PROGRAM EM03_Placing2
VAR
	
	//Backbone
	FB_StateMachine_Placing2		: FB_StateManager;
	bFl_RunningMachinePlacing2		: BOOL;
	bFl_SeqReset					: BOOL;
	bFl_Manual						: BOOL;
	CheckStatusPlacing2				: checkstatus;
	AlarmEventHistory				: ARRAY[1..20] OF Alarm_Event_History;
	Placing2_Management				: FB_Placing;
	bFl_Flushing					: BOOL;
	PalletID_Placing2				: PalletID_Name;
	Placing2_ID						: STRING;
	bFl_PalletJammed				: BOOL;
	
	//Motor
	Motor_PalletPlacing2			: MotorManagement;
	bFl_MotorPlacing2				: BOOL;
	Motor_Placing2_Error			: BOOL;
	Motor_Placing2_ErrorID			: UINT;
	bFl_MotorPlacing2_Fwd			: BOOL;
	bFl_MotorPlacing2_Rev			: BOOL;
	bFL_Safety						: BOOL;
	AlarmEventActive				: ARRAY[1..20] OF Alarm_Event_Active;
	CheckAcc						: TON;
END_VAR
VAR // added by the converter: edge detectors and wires of the graphical bodies
    _w1 : BOOL;
END_VAR

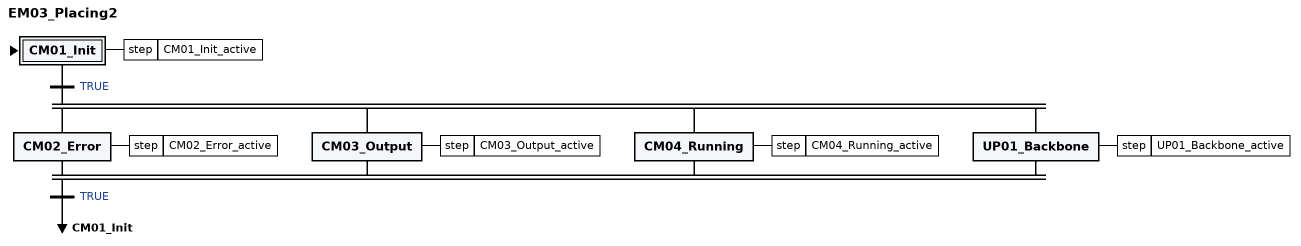
INITIAL_STEP CM01_Init:
    CM01_Init_active(N);  // step action
END_STEP
TRANSITION FROM CM01_Init TO (CM02_Error, CM03_Output, CM04_Running, UP01_Backbone)
    := TRUE;
END_TRANSITION
STEP CM02_Error:
    CM02_Error_active(N);  // step action
END_STEP
STEP CM03_Output:
    CM03_Output_active(N);  // step action
END_STEP
STEP CM04_Running:
    CM04_Running_active(N);  // step action
END_STEP
STEP UP01_Backbone:
    UP01_Backbone_active(N);  // step action
END_STEP
TRANSITION FROM (CM02_Error, CM03_Output, CM04_Running, UP01_Backbone) TO CM01_Init
    := TRUE;
END_TRANSITION

ACTION CM01_Init_active:
Data_GVL.bFL_StartPlacing2			:= Status_GVL.bFl_RunButton_Robotic OR HMI_GVL.bStartButtonPlacing2;
Data_GVL.bFL_StopPlacing2			:= NOT Status_GVL.bFl_StopButton_Robotic OR HMI_GVL.bStopButtonPlacing2;
Data_GVL.bFL_ResetPlacing2			:= Status_GVL.bFl_ResetButton_Robotic OR HMI_GVL.bResetButtonPlacing2;
Data_GVL.bFL_AckPlacing2			:= Status_GVL.bFl_Acknowledge_Robotic OR HMI_GVL.bAcknowledgeButtonPlacing2;
Data_GVL.bFL_AutoManuaModePlacing2 	:= Status_GVL.bFl_Manual_Robotic OR HMI_GVL.bTestModeEnablePlacing2;
bFl_RunningMachinePlacing2			:= Data_GVL.stStateMachinePlacing2.Running;
bFl_Manual							:= Data_GVL.stStateMachinePlacing2.ManualMode;
bFl_SeqReset						:= NOT Status_GVL.bFl_EStop_Robotic;
bFL_Safety							:= Status_GVL.bFl_EStop_Robotic AND Status_GVL.bSafety_DoorRobotic;


(*=================Convert Timer============================*)
Data_GVL.Tmr_Placing2	:= ConvertMilliSecTimeData(HMI_GVL.Tmr_Placing2);

(*=================Data OEE============================*)
Data_GVL.dt_Production[2].Data1			:= HMI_GVL.arCountTotal[2];
Data_GVL.dt_Production[2].Data2			:= HMI_GVL.arPalletTotal[2];
Data_GVL.dt_Production[2].Data3			:= HMI_GVL.arPalletIncomplete[2];
Data_GVL.dt_Production[2].ProductCode	:= Status_GVL.RecipeLine[2].ProductName;
END_ACTION

ACTION CM02_Error_active:
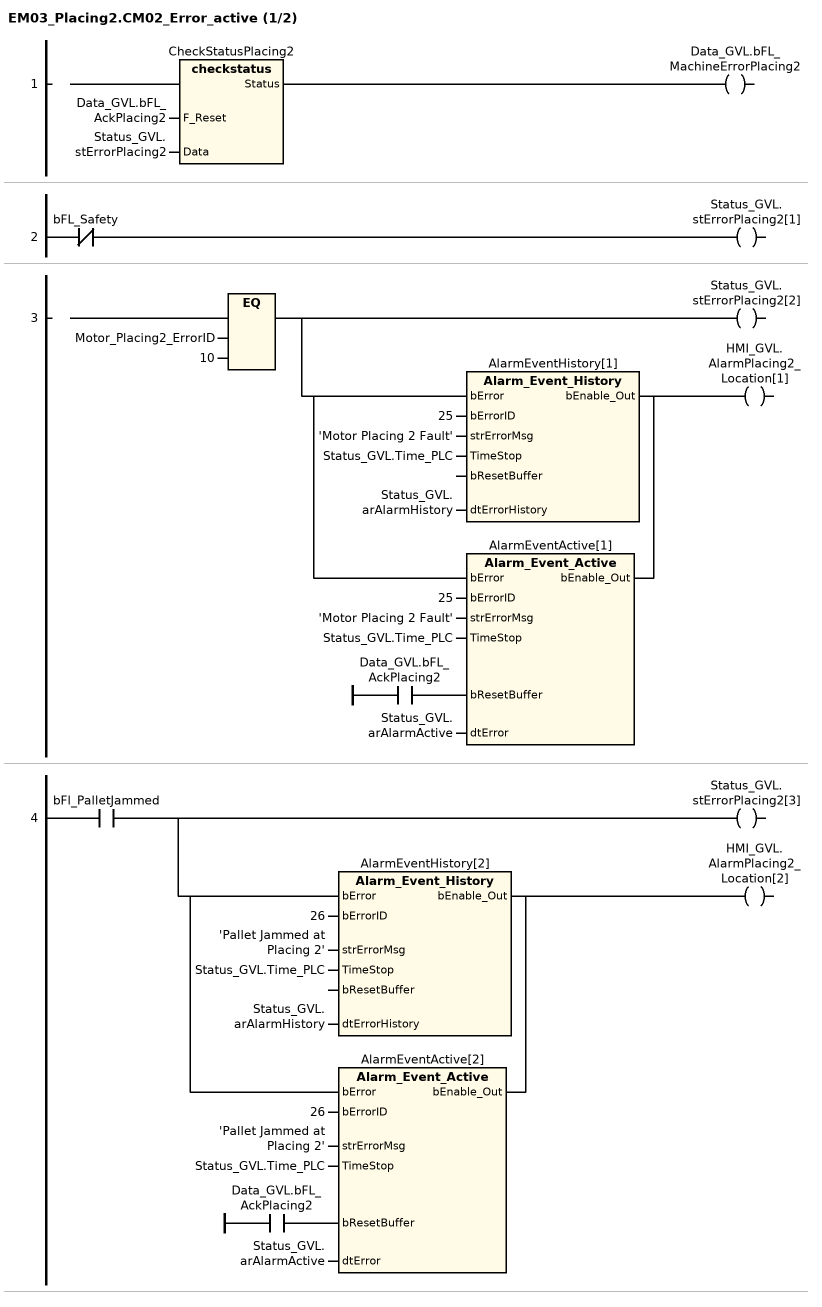
// NETWORK 1
CheckStatusPlacing2(F_Reset := Data_GVL.bFL_AckPlacing2, Data := Status_GVL.stErrorPlacing2); // checkstatus
Data_GVL.bFL_MachineErrorPlacing2 := CheckStatusPlacing2.Status;

// NETWORK 2
Status_GVL.stErrorPlacing2[1] := NOT bFL_Safety;

// NETWORK 3
_w1 := Motor_Placing2_ErrorID = 10;
Status_GVL.stErrorPlacing2[2] := _w1;
AlarmEventHistory[1](
    bError := _w1,
    bErrorID := 25,
    strErrorMsg := 'Motor Placing 2 Fault',
    TimeStop := Status_GVL.Time_PLC,
    dtErrorHistory := Status_GVL.arAlarmHistory); // Alarm_Event_History
AlarmEventActive[1](
    bError := _w1,
    bErrorID := 25,
    strErrorMsg := 'Motor Placing 2 Fault',
    TimeStop := Status_GVL.Time_PLC,
    bResetBuffer := Data_GVL.bFL_AckPlacing2,
    dtError := Status_GVL.arAlarmActive); // Alarm_Event_Active
HMI_GVL.AlarmPlacing2_Location[1] := AlarmEventHistory[1].bEnable_Out OR AlarmEventActive[1].bEnable_Out;

// NETWORK 4
Status_GVL.stErrorPlacing2[3] := bFl_PalletJammed;
AlarmEventHistory[2](
    bError := bFl_PalletJammed,
    bErrorID := 26,
    strErrorMsg := 'Pallet Jammed at Placing 2',
    TimeStop := Status_GVL.Time_PLC,
    dtErrorHistory := Status_GVL.arAlarmHistory); // Alarm_Event_History
AlarmEventActive[2](
    bError := bFl_PalletJammed,
    bErrorID := 26,
    strErrorMsg := 'Pallet Jammed at Placing 2',
    TimeStop := Status_GVL.Time_PLC,
    bResetBuffer := Data_GVL.bFL_AckPlacing2,
    dtError := Status_GVL.arAlarmActive); // Alarm_Event_Active
HMI_GVL.AlarmPlacing2_Location[2] := AlarmEventHistory[2].bEnable_Out OR AlarmEventActive[2].bEnable_Out;

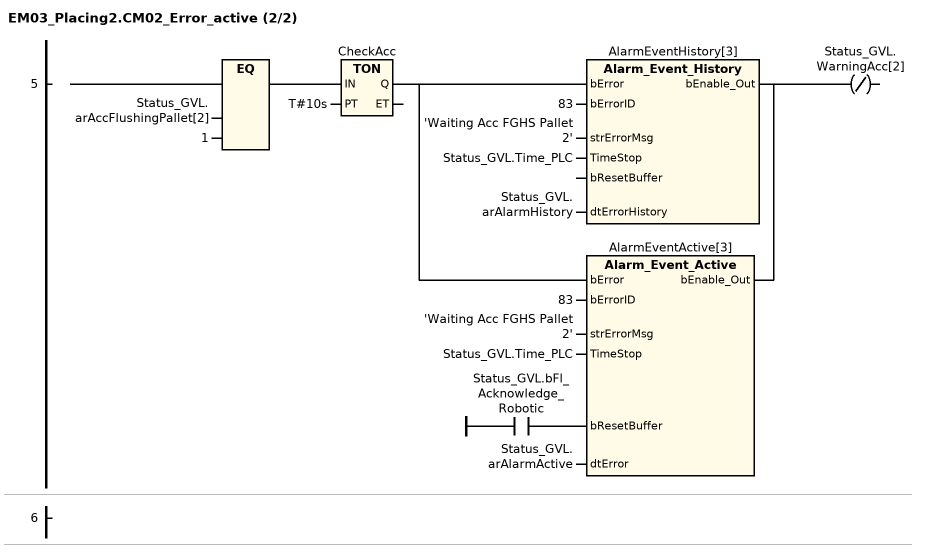
// NETWORK 5
CheckAcc(IN := Status_GVL.arAccFlushingPallet[2] = 1, PT := T#10s); // TON
AlarmEventHistory[3](
    bError := CheckAcc.Q,
    bErrorID := 83,
    strErrorMsg := 'Waiting Acc FGHS Pallet 2',
    TimeStop := Status_GVL.Time_PLC,
    dtErrorHistory := Status_GVL.arAlarmHistory); // Alarm_Event_History
AlarmEventActive[3](
    bError := CheckAcc.Q,
    bErrorID := 83,
    strErrorMsg := 'Waiting Acc FGHS Pallet 2',
    TimeStop := Status_GVL.Time_PLC,
    bResetBuffer := Status_GVL.bFl_Acknowledge_Robotic,
    dtError := Status_GVL.arAlarmActive); // Alarm_Event_Active
Status_GVL.WarningAcc[2] := NOT (AlarmEventHistory[3].bEnable_Out OR AlarmEventActive[3].bEnable_Out);

// NETWORK 6
END_ACTION

ACTION CM03_Output_active:
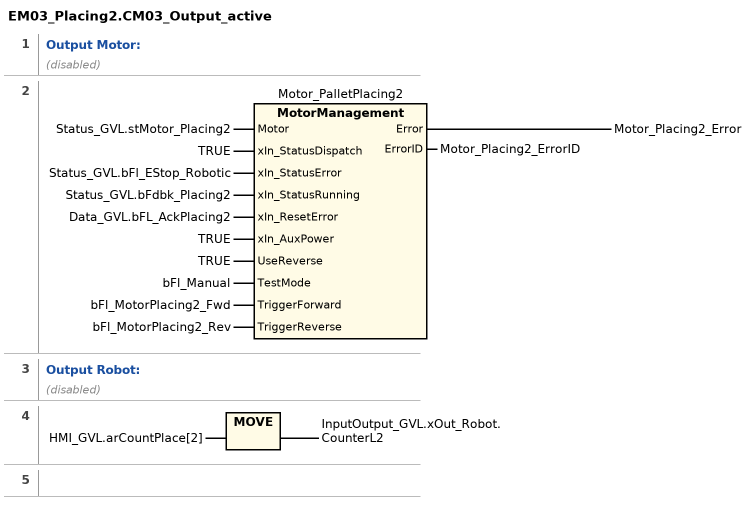
// NETWORK 1 (disabled)
// label: Output Motor

// NETWORK 2
Motor_PalletPlacing2(
    Motor := Status_GVL.stMotor_Placing2,
    xIn_StatusDispatch := TRUE,
    xIn_StatusError := Status_GVL.bFl_EStop_Robotic,
    xIn_StatusRunning := Status_GVL.bFdbk_Placing2,
    xIn_ResetError := Data_GVL.bFL_AckPlacing2,
    xIn_AuxPower := TRUE,
    UseReverse := TRUE,
    TestMode := bFl_Manual,
    TriggerForward := bFl_MotorPlacing2_Fwd,
    TriggerReverse := bFl_MotorPlacing2_Rev,
    ErrorID => Motor_Placing2_ErrorID); // MotorManagement
Motor_Placing2_Error := Motor_PalletPlacing2.Error;

// NETWORK 3 (disabled)
// label: Output Robot

// NETWORK 4
InputOutput_GVL.xOut_Robot.CounterL2 := HMI_GVL.arCountPlace[2];

// NETWORK 5
END_ACTION

ACTION CM04_Running_active:
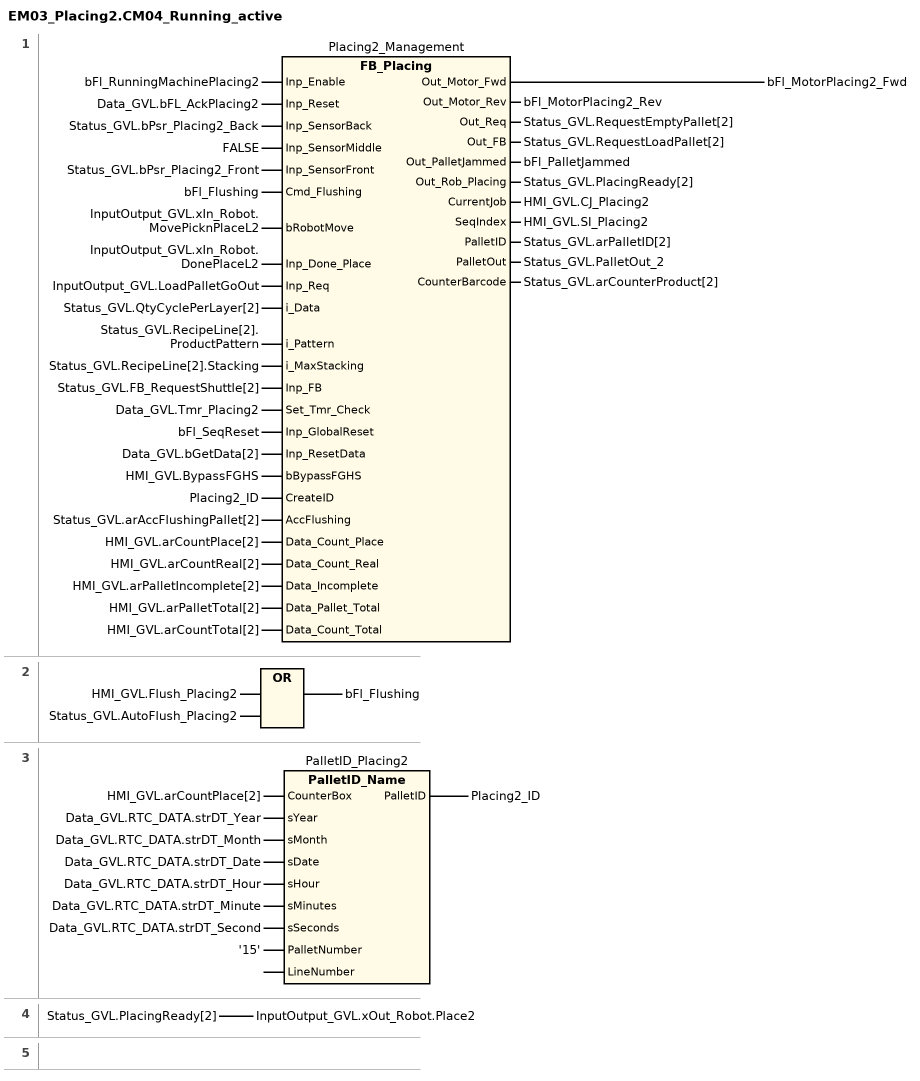
// NETWORK 1
Placing2_Management(
    Inp_Enable := bFl_RunningMachinePlacing2,
    Inp_Reset := Data_GVL.bFL_AckPlacing2,
    Inp_SensorBack := Status_GVL.bPsr_Placing2_Back,
    Inp_SensorMiddle := FALSE,
    Inp_SensorFront := Status_GVL.bPsr_Placing2_Front,
    Cmd_Flushing := bFl_Flushing,
    bRobotMove := InputOutput_GVL.xIn_Robot.MovePicknPlaceL2,
    Inp_Done_Place := InputOutput_GVL.xIn_Robot.DonePlaceL2,
    Inp_Req := InputOutput_GVL.LoadPalletGoOut,
    i_Data := Status_GVL.QtyCyclePerLayer[2],
    i_Pattern := Status_GVL.RecipeLine[2].ProductPattern,
    i_MaxStacking := Status_GVL.RecipeLine[2].Stacking,
    Inp_FB := Status_GVL.FB_RequestShuttle[2],
    Set_Tmr_Check := Data_GVL.Tmr_Placing2,
    Inp_GlobalReset := bFl_SeqReset,
    Inp_ResetData := Data_GVL.bGetData[2],
    bBypassFGHS := HMI_GVL.BypassFGHS,
    CreateID := Placing2_ID,
    AccFlushing := Status_GVL.arAccFlushingPallet[2],
    Data_Count_Place := HMI_GVL.arCountPlace[2],
    Data_Count_Real := HMI_GVL.arCountReal[2],
    Data_Incomplete := HMI_GVL.arPalletIncomplete[2],
    Data_Pallet_Total := HMI_GVL.arPalletTotal[2],
    Data_Count_Total := HMI_GVL.arCountTotal[2],
    Out_Motor_Rev => bFl_MotorPlacing2_Rev,
    Out_Req => Status_GVL.RequestEmptyPallet[2],
    Out_FB => Status_GVL.RequestLoadPallet[2],
    Out_PalletJammed => bFl_PalletJammed,
    Out_Rob_Placing => Status_GVL.PlacingReady[2],
    CurrentJob => HMI_GVL.CJ_Placing2,
    SeqIndex => HMI_GVL.SI_Placing2,
    PalletID => Status_GVL.arPalletID[2],
    PalletOut => Status_GVL.PalletOut_2,
    CounterBarcode => Status_GVL.arCounterProduct[2]); // FB_Placing
bFl_MotorPlacing2_Fwd := Placing2_Management.Out_Motor_Fwd;

// NETWORK 2
bFl_Flushing := HMI_GVL.Flush_Placing2 OR Status_GVL.AutoFlush_Placing2;

// NETWORK 3
PalletID_Placing2(
    CounterBox := HMI_GVL.arCountPlace[2],
    sYear := Data_GVL.RTC_DATA.strDT_Year,
    sMonth := Data_GVL.RTC_DATA.strDT_Month,
    sDate := Data_GVL.RTC_DATA.strDT_Date,
    sHour := Data_GVL.RTC_DATA.strDT_Hour,
    sMinutes := Data_GVL.RTC_DATA.strDT_Minute,
    sSeconds := Data_GVL.RTC_DATA.strDT_Second,
    PalletNumber := '15'); // PalletID_Name
Placing2_ID := PalletID_Placing2.PalletID;

// NETWORK 4
InputOutput_GVL.xOut_Robot.Place2 := Status_GVL.PlacingReady[2];

// NETWORK 5
END_ACTION

ACTION UP01_Backbone_active:
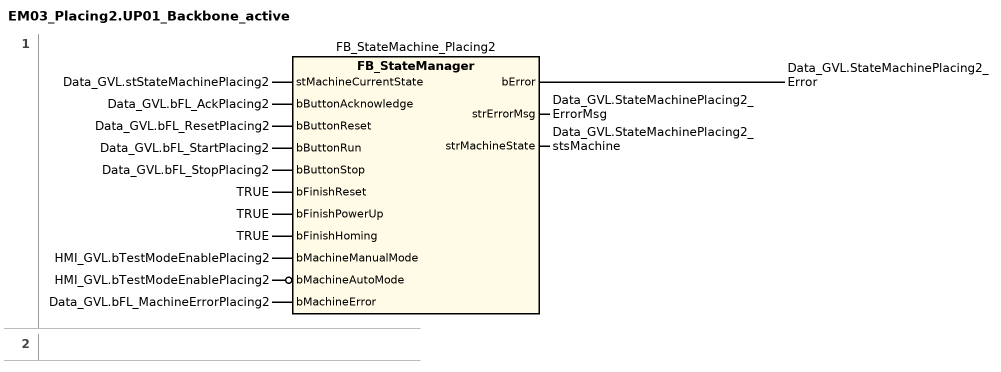
// NETWORK 1
FB_StateMachine_Placing2(
    stMachineCurrentState := Data_GVL.stStateMachinePlacing2,
    bButtonAcknowledge := Data_GVL.bFL_AckPlacing2,
    bButtonReset := Data_GVL.bFL_ResetPlacing2,
    bButtonRun := Data_GVL.bFL_StartPlacing2,
    bButtonStop := Data_GVL.bFL_StopPlacing2,
    bFinishReset := TRUE,
    bFinishPowerUp := TRUE,
    bFinishHoming := TRUE,
    bMachineManualMode := HMI_GVL.bTestModeEnablePlacing2,
    bMachineAutoMode := NOT HMI_GVL.bTestModeEnablePlacing2,
    bMachineError := Data_GVL.bFL_MachineErrorPlacing2,
    strErrorMsg => Data_GVL.StateMachinePlacing2_ErrorMsg,
    strMachineState => Data_GVL.StateMachinePlacing2_stsMachine); // FB_StateManager
Data_GVL.StateMachinePlacing2_Error := FB_StateMachine_Placing2.bError;

// NETWORK 2
END_ACTION

END_PROGRAM

(* stored: Version 1.1.0.1, ProductVersion 3.1.4024.12
   POU EM03_Placing2: Id {fd45ecf3-af2c-4dcd-9a4e-6d724b51984a}, SpecialFunc None
   Action CM01_Init_active: Id {67052a7c-6bb4-4805-b494-30d79d49c686}
   Action CM02_Error_active: Id {6aa11972-4366-4665-aaed-78e83ed1b747}
   Action CM03_Output_active: Id {aca06a9f-918c-403d-ab6c-f9e443ef4b99}
   Action CM04_Running_active: Id {0b7e16bf-2eb8-4daf-8f68-7dd7b02b5839}
   Action UP01_Backbone_active: Id {79260e68-1018-4cca-8c94-3e064b77f1c1} *)
